// TwinCAT 3 PLC project sample_delivery
// ProgramVersion: 3.1.4023.0
// libraries:
//   LCLS Sample Delivery, * (SLAC - LCLS)
//   LCLS Vacuum, * (SLAC - LCLS)
//   Tc2_Standard, * (Beckhoff Automation GmbH)
//   Tc2_System, * (Beckhoff Automation GmbH)
//   Tc3_Module, * (Beckhoff Automation GmbH)
// project tree:
//   GVLs/ GVL_RCC.TcGVL (not stored), GVL_SDS.TcGVL
//   / PlcTask.TcTTO (not stored), SerialComm.TcTTO (not stored)
//   POUs/ MAIN.TcPOU (not stored), PRG_RCC.TcPOU, SerialTxRx.TcPOU (not stored)
// real-time tasks:
//   TASK PlcTask: cycle T#10ms, priority 20, ADS port 350
//   TASK SerialComm: cycle T#10ms, priority 1, ADS port 351
// I/O:
//   DEVICE Device 1 (EtherCAT), AmsNetId 172.21.38.25.2.1
//     Term 1 (EK1200)
//     Box 17 (EP9128-0021)
//     ALI (EP1111)
//     ALI_X (EP7041-0002)
//     ALI_Y (EP7041-0002)
//     ALI_Z (EP7041-0002)
//     ALI_X_ENC (EP5101-0011)
//     ALI_Gauges (EP3174-0002)
//     ALI_PropValve (EP7041-0002)
//     ALI_Y_ENC (EP5101-0011)
//     ALI_DIO (EP2338-0001)
//     M3 Selector A (EP1111)
//     M3 Selector A Digital IO (EP2338-1001)
//     M3 Selector A Serial IO (EP6002-0002)
//     M3 Selector B (EP1111)
//     M3 Selector B Digital IO (EP2338-1001)
//     M3 Selector B Serial IO (EP6002-0002)
//     PCM A (EP1111)
//     PCM A (EP4374-0002)
//     PCM A (EP3174-0002)
//     PCM A (EP6002-0002)
//     PCM B (EP1111)
//     PCM B (EP4374-0002)
//     PCM B (EP3174-0002)
//     PCM B (EP6002-0002)
//     Gas_Mani (EP1111)
//     Gas_Mani_NeedleValve (EP4374-0002)
//     Gas_Mani_ValveCtrl (EP2338-0001)
//     Gas_Mani_ValveRbk (EP2338-0001)
//     M3 Selector C (EP1111)
//     M3 Selector C Digital IO (EP2338-1001)
//     M3 Selector C Serial IO (EP6002-0002)
//     M3 Selector D (EP1111)
//     M3 Selector D Digital IO (EP2338-1001)
//     M3 Selector D Serial IO (EP6002-0002)
//     PCM C (EP1111)
//     PCM C (EP4374-0002)
//     PCM C (EP3174-0002)
//     PCM C (EP6002-0002)
//     PCM D (EP1111)
//     PCM D (EP4374-0002)
//     PCM D (EP3174-0002)
//     PCM D (EP6002-0002)
//     Bronkhorst MFM A
//     Bronkhorst MFM B
//     Bronkhorst MFM C
//     Bronkhorst MFM D
//     Solenoid Pair A (EP1111)
//     Solenoid Pair A Digital IO (EP2338-0001)
//     RCC A (EP1111)
//     RCC (EP2338-0001)
//     RCC_PCM_A (EP4374-0002) [EP4374-0002 2Ch. Ana. Input +/-10V, 0-10V, 0/4-20mA configurable; 2Ch. Ana. Output +/-10V, 0-10V, 0/4-20mA configurable]
// variable links:
//   sample-delivery Instance <-> Device 1 (EtherCAT)/Bronkhorst MFM A
//     PlcTask Inputs/GVL_SDS.BronkhorstA.stMFM.i_rFlow <-> TxPDO Map/fMeasure
//     PlcTask Outputs/GVL_SDS.BronkhorstA.stMFM.q_rSetpoint <-> RxPDO Map/fSetpoint
//   sample-delivery Instance <-> Device 1 (EtherCAT)/Bronkhorst MFM B
//     PlcTask Inputs/GVL_SDS.BronkhorstB.stMFM.i_rFlow <-> TxPDO Map/fMeasure
//     PlcTask Outputs/GVL_SDS.BronkhorstB.stMFM.q_rSetpoint <-> RxPDO Map/fSetpoint
//   sample-delivery Instance <-> Device 1 (EtherCAT)/Gas_Mani_ValveCtrl (EP2338-0001)
//     PlcTask Outputs/GVL_SDS.GasMan.stValve[{1..7}].qxDO <-> Channel {9..15}/Output  (7 links)
//   sample-delivery Instance <-> Device 1 (EtherCAT)/Gas_Mani_ValveRbk (EP2338-0001)
//     PlcTask Inputs/GVL_SDS.GasMan.stValve[{1..7}].ixOPN <-> Channel {1..7}/Input  (7 links)
//   sample-delivery Instance <-> Device 1 (EtherCAT)/M3 Selector A Digital IO (EP2338-1001)
//     PlcTask Outputs/GVL_SDS.M3SelectorA.stShaker01.q_xPwrDO <-> Channel 9/Output
//     PlcTask Outputs/GVL_SDS.M3SelectorA.stShaker02.q_xPwrDO <-> Channel 10/Output
//     PlcTask Outputs/GVL_SDS.M3SelectorA.stShaker03.q_xPwrDO <-> Channel 11/Output
//     PlcTask Outputs/GVL_SDS.M3SelectorA.stShaker04.q_xPwrDO <-> Channel 12/Output
//   sample-delivery Instance <-> Device 1 (EtherCAT)/M3 Selector A Serial IO (EP6002-0002)
//     SerialComm Inputs/GVL_SDS.M3SelectorA.stSensSerial.stComIn/Status <-> COM TxPDO-Map Inputs Channel 1/Status
//     SerialComm Inputs/GVL_SDS.M3SelectorA.stViciSerial.stComIn/Status <-> COM TxPDO-Map Inputs Channel 2/Status
//   sample-delivery Instance <-> Device 1 (EtherCAT)/M3 Selector B Digital IO (EP2338-1001)
//     PlcTask Outputs/GVL_SDS.M3SelectorB.stShaker01.q_xPwrDO <-> Channel 9/Output
//     PlcTask Outputs/GVL_SDS.M3SelectorB.stShaker02.q_xPwrDO <-> Channel 10/Output
//     PlcTask Outputs/GVL_SDS.M3SelectorB.stShaker03.q_xPwrDO <-> Channel 11/Output
//     PlcTask Outputs/GVL_SDS.M3SelectorB.stShaker04.q_xPwrDO <-> Channel 12/Output
//   sample-delivery Instance <-> Device 1 (EtherCAT)/M3 Selector B Serial IO (EP6002-0002)
//     SerialComm Inputs/GVL_SDS.M3SelectorB.stSensSerial.stComIn/Status <-> COM TxPDO-Map Inputs Channel 1/Status
//     SerialComm Inputs/GVL_SDS.M3SelectorB.stViciSerial.stComIn/Status <-> COM TxPDO-Map Inputs Channel 2/Status
//   sample-delivery Instance <-> Device 1 (EtherCAT)/M3 Selector C Digital IO (EP2338-1001)
//     PlcTask Outputs/GVL_SDS.M3SelectorC.stShaker01.q_xPwrDO <-> Channel 9/Output
//     PlcTask Outputs/GVL_SDS.M3SelectorC.stShaker02.q_xPwrDO <-> Channel 10/Output
//     PlcTask Outputs/GVL_SDS.M3SelectorC.stShaker03.q_xPwrDO <-> Channel 11/Output
//     PlcTask Outputs/GVL_SDS.M3SelectorC.stShaker04.q_xPwrDO <-> Channel 12/Output
//   sample-delivery Instance <-> Device 1 (EtherCAT)/M3 Selector C Serial IO (EP6002-0002)
//     SerialComm Inputs/GVL_SDS.M3SelectorC.stSensSerial.stComIn/Status <-> COM TxPDO-Map Inputs Channel 1/Status
//     SerialComm Inputs/GVL_SDS.M3SelectorC.stViciSerial.stComIn/Status <-> COM TxPDO-Map Inputs Channel 2/Status
//   sample-delivery Instance <-> Device 1 (EtherCAT)/M3 Selector D Digital IO (EP2338-1001)
//     PlcTask Outputs/GVL_SDS.M3SelectorD.stShaker01.q_xPwrDO <-> Channel 9/Output
//     PlcTask Outputs/GVL_SDS.M3SelectorD.stShaker02.q_xPwrDO <-> Channel 10/Output
//     PlcTask Outputs/GVL_SDS.M3SelectorD.stShaker03.q_xPwrDO <-> Channel 11/Output
//     PlcTask Outputs/GVL_SDS.M3SelectorD.stShaker04.q_xPwrDO <-> Channel 12/Output
//   sample-delivery Instance <-> Device 1 (EtherCAT)/M3 Selector D Serial IO (EP6002-0002)
//     SerialComm Inputs/GVL_SDS.M3SelectorD.stSensSerial.stComIn/Status <-> COM TxPDO-Map Inputs Channel 1/Status
//     SerialComm Inputs/GVL_SDS.M3SelectorD.stViciSerial.stComIn/Status <-> COM TxPDO-Map Inputs Channel 2/Status
//   sample-delivery Instance <-> Device 1 (EtherCAT)/PCM A (EP1111)
//     PlcTask Inputs/GVL_SDS.PCMA.stBaseIO.i_SyncUnitWC <-> WcState/WcState
//   sample-delivery Instance <-> Device 1 (EtherCAT)/PCM A (EP4374-0002)
//     PlcTask Inputs/GVL_SDS.PCMA.stPropAir1.i_iPressRB <-> AI Inputs Channel 1/Value
//     PlcTask Inputs/GVL_SDS.PCMA.stPropAir2.i_iPressRB <-> AI Inputs Channel 2/Value
//     PlcTask Outputs/GVL_SDS.PCMA.stPropAir1.q_iPressCt <-> AO Outputs Channel 3/Analog output
//     PlcTask Outputs/GVL_SDS.PCMA.stPropAir2.q_iPressCt <-> AO Outputs Channel 4/Analog output
//   sample-delivery Instance <-> Device 1 (EtherCAT)/PCM A (EP6002-0002)
//     SerialComm Inputs/GVL_SDS.PCMA.stSerial1.stComIn/Status <-> COM TxPDO-Map Inputs Channel 1/Status
//     SerialComm Inputs/GVL_SDS.PCMA.stSerial2.stComIn/Status <-> COM TxPDO-Map Inputs Channel 2/Status
//     SerialComm Outputs/GVL_SDS.PCMA.stSerial1.stComOut/Ctrl <-> COM RxPDO-Map Outputs Channel 1/Ctrl
//     SerialComm Outputs/GVL_SDS.PCMA.stSerial2.stComOut/Ctrl <-> COM RxPDO-Map Outputs Channel 2/Ctrl
//   sample-delivery Instance <-> Device 1 (EtherCAT)/PCM B (EP1111)
//     PlcTask Inputs/GVL_SDS.PCMB.stBaseIO.i_SyncUnitWC <-> WcState/WcState
//   sample-delivery Instance <-> Device 1 (EtherCAT)/PCM B (EP4374-0002)
//     PlcTask Inputs/GVL_SDS.PCMB.stPropAir1.i_iPressRB <-> AI Inputs Channel 1/Value
//     PlcTask Inputs/GVL_SDS.PCMB.stPropAir2.i_iPressRB <-> AI Inputs Channel 2/Value
//     PlcTask Outputs/GVL_SDS.PCMB.stPropAir1.q_iPressCt <-> AO Outputs Channel 3/Analog output
//     PlcTask Outputs/GVL_SDS.PCMB.stPropAir2.q_iPressCt <-> AO Outputs Channel 4/Analog output
//   sample-delivery Instance <-> Device 1 (EtherCAT)/PCM B (EP6002-0002)
//     SerialComm Inputs/GVL_SDS.PCMB.stSerial1.stComIn/Status <-> COM TxPDO-Map Inputs Channel 1/Status
//     SerialComm Inputs/GVL_SDS.PCMB.stSerial2.stComIn/Status <-> COM TxPDO-Map Inputs Channel 2/Status
//     SerialComm Outputs/GVL_SDS.PCMB.stSerial1.stComOut/Ctrl <-> COM RxPDO-Map Outputs Channel 1/Ctrl
//     SerialComm Outputs/GVL_SDS.PCMB.stSerial2.stComOut/Ctrl <-> COM RxPDO-Map Outputs Channel 2/Ctrl
//   sample-delivery Instance <-> Device 1 (EtherCAT)/PCM C (EP1111)
//     PlcTask Inputs/GVL_SDS.PCMC.stBaseIO.i_SyncUnitWC <-> WcState/WcState
//   sample-delivery Instance <-> Device 1 (EtherCAT)/PCM C (EP4374-0002)
//     PlcTask Inputs/GVL_SDS.PCMC.stPropAir1.i_iPressRB <-> AI Inputs Channel 1/Value
//     PlcTask Inputs/GVL_SDS.PCMC.stPropAir2.i_iPressRB <-> AI Inputs Channel 2/Value
//     PlcTask Outputs/GVL_SDS.PCMC.stPropAir1.q_iPressCt <-> AO Outputs Channel 3/Analog output
//     PlcTask Outputs/GVL_SDS.PCMC.stPropAir2.q_iPressCt <-> AO Outputs Channel 4/Analog output
//   sample-delivery Instance <-> Device 1 (EtherCAT)/PCM C (EP6002-0002)
//     SerialComm Inputs/GVL_SDS.PCMC.stSerial1.stComIn/Status <-> COM TxPDO-Map Inputs Channel 1/Status
//     SerialComm Inputs/GVL_SDS.PCMC.stSerial2.stComIn/Status <-> COM TxPDO-Map Inputs Channel 2/Status
//     SerialComm Outputs/GVL_SDS.PCMC.stSerial1.stComOut/Ctrl <-> COM RxPDO-Map Outputs Channel 1/Ctrl
//     SerialComm Outputs/GVL_SDS.PCMC.stSerial2.stComOut/Ctrl <-> COM RxPDO-Map Outputs Channel 2/Ctrl
//   sample-delivery Instance <-> Device 1 (EtherCAT)/PCM D (EP1111)
//     PlcTask Inputs/GVL_SDS.PCMD.stBaseIO.i_SyncUnitWC <-> WcState/WcState
//   sample-delivery Instance <-> Device 1 (EtherCAT)/PCM D (EP4374-0002)
//     PlcTask Inputs/GVL_SDS.PCMD.stPropAir1.i_iPressRB <-> AI Inputs Channel 1/Value
//     PlcTask Inputs/GVL_SDS.PCMD.stPropAir2.i_iPressRB <-> AI Inputs Channel 2/Value
//     PlcTask Outputs/GVL_SDS.PCMD.stPropAir1.q_iPressCt <-> AO Outputs Channel 3/Analog output
//     PlcTask Outputs/GVL_SDS.PCMD.stPropAir2.q_iPressCt <-> AO Outputs Channel 4/Analog output
//   sample-delivery Instance <-> Device 1 (EtherCAT)/PCM D (EP6002-0002)
//     SerialComm Inputs/GVL_SDS.PCMD.stSerial1.stComIn/Status <-> COM TxPDO-Map Inputs Channel 1/Status
//     SerialComm Inputs/GVL_SDS.PCMD.stSerial2.stComIn/Status <-> COM TxPDO-Map Inputs Channel 2/Status
//     SerialComm Outputs/GVL_SDS.PCMD.stSerial1.stComOut/Ctrl <-> COM RxPDO-Map Outputs Channel 1/Ctrl
//     SerialComm Outputs/GVL_SDS.PCMD.stSerial2.stComOut/Ctrl <-> COM RxPDO-Map Outputs Channel 2/Ctrl
//   sample-delivery Instance <-> Device 1 (EtherCAT)/RCC (EP2338-0001)
//     PlcTask Inputs/GVL_RCC.RCC_VRC_01.i_xOpnLS <-> Channel 1/Input
//     PlcTask Inputs/GVL_RCC.RCC_VRC_02.i_xOpnLS <-> Channel 2/Input
//     PlcTask Inputs/GVL_RCC.RCC_VRC_03.i_xOpnLS <-> Channel 3/Input
//     PlcTask Inputs/GVL_RCC.RCC_VRC_04.i_xOpnLS <-> Channel 4/Input
//     PlcTask Inputs/GVL_RCC.RCC_VRC_05.i_xOpnLS <-> Channel 5/Input
//     PlcTask Inputs/GVL_RCC.RCC_VRC_06.i_xOpnLS <-> Channel 6/Input
//     PlcTask Inputs/GVL_RCC.RCC_VRC_07.i_xOpnLS <-> Channel 7/Input
//     PlcTask Inputs/GVL_RCC.RCC_VRC_08.i_xOpnLS <-> Channel 8/Input
//     PlcTask Outputs/GVL_RCC.RCC_VRC_01.q_xOPN_DO <-> Channel 9/Output
//     PlcTask Outputs/GVL_RCC.RCC_VRC_02.q_xOPN_DO <-> Channel 10/Output
//     PlcTask Outputs/GVL_RCC.RCC_VRC_03.q_xOPN_DO <-> Channel 11/Output
//     PlcTask Outputs/GVL_RCC.RCC_VRC_04.q_xOPN_DO <-> Channel 12/Output
//     PlcTask Outputs/GVL_RCC.RCC_VRC_05.q_xOPN_DO <-> Channel 13/Output
//     PlcTask Outputs/GVL_RCC.RCC_VRC_06.q_xOPN_DO <-> Channel 14/Output
//     PlcTask Outputs/GVL_RCC.RCC_VRC_07.q_xOPN_DO <-> Channel 15/Output
//     PlcTask Outputs/GVL_RCC.RCC_VRC_08.q_xOPN_DO <-> Channel 16/Output
//   sample-delivery Instance <-> Device 1 (EtherCAT)/RCC_PCM_A (EP4374-0002)
//     PlcTask Inputs/PRG_RCC.RCC_PCM.stPropAir1.i_iPressRB <-> AI Inputs Channel 1/Value
//     PlcTask Inputs/PRG_RCC.RCC_PCM.stPropAir2.i_iPressRB <-> AI Inputs Channel 2/Value
//     PlcTask Outputs/PRG_RCC.RCC_PCM.stPropAir1.q_iPressCt <-> AO Outputs Channel 3/Analog output
//     PlcTask Outputs/PRG_RCC.RCC_PCM.stPropAir2.q_iPressCt <-> AO Outputs Channel 4/Analog output
//   sample-delivery Instance <-> Device 1 (EtherCAT)/Solenoid Pair A Digital IO (EP2338-0001)
//     PlcTask Outputs/GVL_SDS.SolenoidPairA.q_xDO1 <-> Channel 9/Output
//     PlcTask Outputs/GVL_SDS.SolenoidPairA.q_xDO2 <-> Channel 10/Output

// ---- GVLs/GVL_SDS.TcGVL
VAR_GLOBAL

// TODO: FIX Linking for Devices will be deployed
//  Working: Bronkhorst MFM B
{attribute 'pytmc' := 'pv: XCS:SDS:SEL:A'}
{attribute 'TcLinkTo' := '.stSensSerial.stComIn.Status := TIIB[M3 Selector A Serial IO (EP6002-0002)]^COM TxPDO-Map Inputs Channel 1^Status;
                          .stViciSerial.stComIn.Status := TIIB[M3 Selector A Serial IO (EP6002-0002)]^COM TxPDO-Map Inputs Channel 2^Status;
                          .stSensSerial.stComOut.Ctrl := TIID^MAIN (EtherCAT)^M3 Selector A Serial IO (EP6002-0002)^COM RxPDO-Map Outputs Channel 1^Ctrl;
                          .stViciSerial.stComOut.Ctrl := TIID^MAIN (EtherCAT)^M3 Selector A Serial IO (EP6002-0002)^COM RxPDO-Map Outputs Channel 2^Ctrl;
                          .stShaker01.q_xPwrDO := TIIB[M3 Selector A Digital IO (EP2338-1001)]^Channel 9^Output;
                          .stShaker02.q_xPwrDO := TIIB[M3 Selector A Digital IO (EP2338-1001)]^Channel 10^Output;
                          .stShaker03.q_xPwrDO := TIIB[M3 Selector A Digital IO (EP2338-1001)]^Channel 11^Output;
                          .stShaker04.q_xPwrDO := TIIB[M3 Selector A Digital IO (EP2338-1001)]^Channel 12^Output;
                          .stBaseIO.i_SyncUnitWC := TIID^MAIN (EtherCAT)^M3 Selector A (EP1111)^WcState^WcState;
                          .
'}
M3SelectorA : FB_SelectorM3;

{attribute 'pytmc' := 'pv: XCS:SDS:SEL:B'}
{attribute 'TcLinkTo' := '.stSensSerial.stComIn.Status := TIIB[M3 Selector B Serial IO (EP6002-0002)]^COM TxPDO-Map Inputs Channel 1^Status;
                          .stViciSerial.stComIn.Status := TIIB[M3 Selector B Serial IO (EP6002-0002)]^COM TxPDO-Map Inputs Channel 2^Status;
                          .stSensSerial.stComOut.Ctrl := TIID^MAIN (EtherCAT)^M3 Selector B Serial IO (EP6002-0002)^COM RxPDO-Map Outputs Channel 1^Ctrl;
                          .stViciSerial.stComOut.Ctrl := TIID^MAIN (EtherCAT)^M3 Selector B Serial IO (EP6002-0002)^COM RxPDO-Map Outputs Channel 2^Ctrl;
                          .stShaker01.q_xPwrDO := TIIB[M3 Selector B Digital IO (EP2338-1001)]^Channel 9^Output;
                          .stShaker02.q_xPwrDO := TIIB[M3 Selector B Digital IO (EP2338-1001)]^Channel 10^Output;
                          .stShaker03.q_xPwrDO := TIIB[M3 Selector B Digital IO (EP2338-1001)]^Channel 11^Output;
                          .stShaker04.q_xPwrDO := TIIB[M3 Selector B Digital IO (EP2338-1001)]^Channel 12^Output;
                          .stBaseIO.i_SyncUnitWC := TIID^MAIN (EtherCAT)^M3 Selector B (EP1111)^WcState^WcState
'}
M3SelectorB : FB_SelectorM3;

{attribute 'pytmc' := 'pv: XCS:SDS:SEL:C'}
{attribute 'TcLinkTo' := '.stSensSerial.stComIn.Status := TIIB[M3 Selector C Serial IO (EP6002-0002)]^COM TxPDO-Map Inputs Channel 1^Status;
                          .stViciSerial.stComIn.Status := TIIB[M3 Selector C Serial IO (EP6002-0002)]^COM TxPDO-Map Inputs Channel 2^Status;
                          .stSensSerial.stComOut.Ctrl := TIID^MAIN (EtherCAT)^M3 Selector C Serial IO (EP6002-0002)^COM RxPDO-Map Outputs Channel 1^Ctrl;
                          .stViciSerial.stComOut.Ctrl := TIID^MAIN (EtherCAT)^M3 Selector C Serial IO (EP6002-0002)^COM RxPDO-Map Outputs Channel 2^Ctrl;
                          .stShaker01.q_xPwrDO := TIIB[M3 Selector C Digital IO (EP2338-1001)]^Channel 9^Output;
                          .stShaker02.q_xPwrDO := TIIB[M3 Selector C Digital IO (EP2338-1001)]^Channel 10^Output;
                          .stShaker03.q_xPwrDO := TIIB[M3 Selector C Digital IO (EP2338-1001)]^Channel 11^Output;
                          .stShaker04.q_xPwrDO := TIIB[M3 Selector C Digital IO (EP2338-1001)]^Channel 12^Output;
                          .stBaseIO.i_SyncUnitWC := TIID^MAIN (EtherCAT)^M3 Selector C (EP1111)^WcState^WcState
'}
M3SelectorC : FB_SelectorM3;

{attribute 'pytmc' := 'pv: XCS:SDS:SEL:D'}
{attribute 'TcLinkTo' := '.stSensSerial.stComIn.Status := TIIB[M3 Selector D Serial IO (EP6002-0002)]^COM TxPDO-Map Inputs Channel 1^Status;
                          .stViciSerial.stComIn.Status := TIIB[M3 Selector D Serial IO (EP6002-0002)]^COM TxPDO-Map Inputs Channel 2^Status;
                          .stSensSerial.stComOut.Ctrl := TIID^MAIN (EtherCAT)^M3 Selector D Serial IO (EP6002-0002)^COM RxPDO-Map Outputs Channel 1^Ctrl;
                          .stViciSerial.stComOut.Ctrl := TIID^MAIN (EtherCAT)^M3 Selector D Serial IO (EP6002-0002)^COM RxPDO-Map Outputs Channel 2^Ctrl;
                          .stShaker01.q_xPwrDO := TIIB[M3 Selector D Digital IO (EP2338-1001)]^Channel 9^Output;
                          .stShaker02.q_xPwrDO := TIIB[M3 Selector D Digital IO (EP2338-1001)]^Channel 10^Output;
                          .stShaker03.q_xPwrDO := TIIB[M3 Selector D Digital IO (EP2338-1001)]^Channel 11^Output;
                          .stShaker04.q_xPwrDO := TIIB[M3 Selector D Digital IO (EP2338-1001)]^Channel 12^Output;
                          .stBaseIO.i_SyncUnitWC := TIID^MAIN (EtherCAT)^M3 Selector D (EP1111)^WcState^WcState
'}
M3SelectorD : FB_SelectorM3;

{attribute 'pytmc' := 'pv: XCS:SDS:PCM:A'}
{attribute 'TcLinkTo' := '.stPropAir1.i_iPressRB 	:= TIIB[PCM A (EP4374-0002)]^AI Inputs Channel 1^Value;
                          .stPropAir2.i_iPressRB 	:= TIIB[PCM A (EP4374-0002)]^AI Inputs Channel 2^Value;
                          .stPropAir1.q_iPressCt 	:= TIIB[PCM A (EP4374-0002)]^AO Outputs Channel 3^Analog output;
                          .stPropAir2.q_iPressCt 	:= TIIB[PCM A (EP4374-0002)]^AO Outputs Channel 4^Analog output;
                          .stSerial1.stComIn.Status := TIIB[PCM A (EP6002-0002)]^COM TxPDO-Map Inputs Channel 1^Status;
                          .stSerial2.stComIn.Status := TIIB[PCM A (EP6002-0002)]^COM TxPDO-Map Inputs Channel 2^Status;
                          .stSerial1.stComOut.Ctrl 	:= TIIB[PCM A (EP6002-0002)]^COM RxPDO-Map Outputs Channel 1^Ctrl;
                          .stSerial2.stComOut.Ctrl 	:= TIIB[PCM A (EP6002-0002)]^COM RxPDO-Map Outputs Channel 2^Ctrl;
                          .stBaseIO.i_SyncUnitWC 	:= TIIB[PCM A (EP1111)]^WcState^WcState;
'}
PCMA : FB_PressureControlModule;

{attribute 'pytmc' := 'pv: XCS:SDS:PCM:B'}
{attribute 'TcLinkTo' := '.stPropAir1.i_iPressRB 	:= TIIB[PCM B (EP4374-0002)]^AI Inputs Channel 1^Value;
                          .stPropAir2.i_iPressRB 	:= TIIB[PCM B (EP4374-0002)]^AI Inputs Channel 2^Value;
                          .stPropAir1.q_iPressCt 	:= TIIB[PCM B (EP4374-0002)]^AO Outputs Channel 3^Analog output;
                          .stPropAir2.q_iPressCt 	:= TIIB[PCM B (EP4374-0002)]^AO Outputs Channel 4^Analog output;
                          .stSerial1.stComIn.Status := TIIB[PCM B (EP6002-0002)]^COM TxPDO-Map Inputs Channel 1^Status;
                          .stSerial2.stComIn.Status := TIIB[PCM B (EP6002-0002)]^COM TxPDO-Map Inputs Channel 2^Status;
                          .stSerial1.stComOut.Ctrl 	:= TIIB[PCM B (EP6002-0002)]^COM RxPDO-Map Outputs Channel 1^Ctrl;
                          .stSerial2.stComOut.Ctrl 	:= TIIB[PCM B (EP6002-0002)]^COM RxPDO-Map Outputs Channel 2^Ctrl;
                          .stBaseIO.i_SyncUnitWC 	:= TIIB[PCM B (EP1111)]^WcState^WcState;
'}
PCMB : FB_PressureControlModule;

{attribute 'pytmc' := 'pv: XCS:SDS:PCM:C'}
{attribute 'TcLinkTo' := '.stPropAir1.i_iPressRB 	:= TIIB[PCM C (EP4374-0002)]^AI Inputs Channel 1^Value;
                          .stPropAir2.i_iPressRB 	:= TIIB[PCM C (EP4374-0002)]^AI Inputs Channel 2^Value;
                          .stPropAir1.q_iPressCt 	:= TIIB[PCM C (EP4374-0002)]^AO Outputs Channel 3^Analog output;
                          .stPropAir2.q_iPressCt 	:= TIIB[PCM C (EP4374-0002)]^AO Outputs Channel 4^Analog output;
                          .stSerial1.stComIn.Status := TIIB[PCM C (EP6002-0002)]^COM TxPDO-Map Inputs Channel 1^Status;
                          .stSerial2.stComIn.Status := TIIB[PCM C (EP6002-0002)]^COM TxPDO-Map Inputs Channel 2^Status;
                          .stSerial1.stComOut.Ctrl 	:= TIIB[PCM C (EP6002-0002)]^COM RxPDO-Map Outputs Channel 1^Ctrl;
                          .stSerial2.stComOut.Ctrl 	:= TIIB[PCM C (EP6002-0002)]^COM RxPDO-Map Outputs Channel 2^Ctrl;
                          .stBaseIO.i_SyncUnitWC 	:= TIIB[PCM C (EP1111)]^WcState^WcState;
                          '}
PCMC : FB_PressureControlModule;

{attribute 'pytmc' := 'pv: XCS:SDS:PCM:D'}
{attribute 'TcLinkTo' := '.stPropAir1.i_iPressRB 	:= TIIB[PCM D (EP4374-0002)]^AI Inputs Channel 1^Value;
                          .stPropAir2.i_iPressRB 	:= TIIB[PCM D (EP4374-0002)]^AI Inputs Channel 2^Value;
                          .stPropAir1.q_iPressCt 	:= TIIB[PCM D (EP4374-0002)]^AO Outputs Channel 3^Analog output;
                          .stPropAir2.q_iPressCt 	:= TIIB[PCM D (EP4374-0002)]^AO Outputs Channel 4^Analog output;
                          .stSerial1.stComIn.Status := TIIB[PCM D (EP6002-0002)]^COM TxPDO-Map Inputs Channel 1^Status;
                          .stSerial2.stComIn.Status := TIIB[PCM D (EP6002-0002)]^COM TxPDO-Map Inputs Channel 2^Status;
                          .stSerial1.stComOut.Ctrl 	:= TIIB[PCM D (EP6002-0002)]^COM RxPDO-Map Outputs Channel 1^Ctrl;
                          .stSerial2.stComOut.Ctrl 	:= TIIB[PCM D (EP6002-0002)]^COM RxPDO-Map Outputs Channel 2^Ctrl;
                          .stBaseIO.i_SyncUnitWC 	:= TIIB[PCM D (EP1111)]^WcState^WcState;
                          '}
PCMD : FB_PressureControlModule;

{attribute 'pytmc' := 'pv: XCS:SDS:MAN'}
{attribute 'TcLinkTo' := '.stValve[1].qxDO := TIIB[Gas_Mani_ValveCtrl (EP2338-0001)]^Channel 9^Output;
                          .stValve[1].ixOPN := TIIB[Gas_Mani_ValveRbk (EP2338-0001)]^Channel 1^Input;
                          .stValve[2].qxDO := TIIB[Gas_Mani_ValveCtrl (EP2338-0001)]^Channel 10^Output;
                          .stValve[2].ixOPN := TIIB[Gas_Mani_ValveRbk (EP2338-0001)]^Channel 2^Input;
                          .stValve[3].qxDO := TIIB[Gas_Mani_ValveCtrl (EP2338-0001)]^Channel 11^Output;
                          .stValve[3].ixOPN := TIIB[Gas_Mani_ValveRbk (EP2338-0001)]^Channel 3^Input;
                          .stValve[4].qxDO := TIIB[Gas_Mani_ValveCtrl (EP2338-0001)]^Channel 12^Output;
                          .stValve[4].ixOPN := TIIB[Gas_Mani_ValveRbk (EP2338-0001)]^Channel 4^Input;
                          .stValve[5].qxDO := TIIB[Gas_Mani_ValveCtrl (EP2338-0001)]^Channel 13^Output;
                          .stValve[5].ixOPN := TIIB[Gas_Mani_ValveRbk (EP2338-0001)]^Channel 5^Input;
                          .stValve[6].qxDO := TIIB[Gas_Mani_ValveCtrl (EP2338-0001)]^Channel 14^Output;
                          .stValve[6].ixOPN := TIIB[Gas_Mani_ValveRbk (EP2338-0001)]^Channel 6^Input;
                          .stValve[7].qxDO := TIIB[Gas_Mani_ValveCtrl (EP2338-0001)]^Channel 15^Output;
                          .stValve[7].ixOPN := TIIB[Gas_Mani_ValveRbk (EP2338-0001)]^Channel 7^Input;
                          .stBaseIO.i_SyncUnitWC :=	TIID^MAIN (EtherCAT)^Gas_Mani (EP1111)^WcState^WcState;
'}
GasMan : FB_GasManifold;

{attribute 'pytmc' := 'pv: XCS:SDS:MFM:A'}
{attribute 'TcLinkTo' := '.stMFM.i_rFlow := 	TIIB[Bronkhorst MFM A]^TxPDO Map^fMeasure;
                          .stMFM.q_rSetpoint := TIIB[Bronkhorst MFM A]^RxPDO Map^fSetpoint;
'}
BronkhorstA : FB_BronkhorstMFM;

{attribute 'pytmc' := 'pv: XCS:SDS:MFM:B'}
{attribute 'TcLinkTo' := '.stMFM.i_rFlow 		:= 	TIIB[Bronkhorst MFM B]^TxPDO Map^fMeasure;
                          .stMFM.q_rSetpoint 	:=  TIIB[Bronkhorst MFM B]^RxPDO Map^fSetpoint;
'}
BronkhorstB : FB_BronkhorstMFM;

{attribute 'pytmc' := 'pv: XCS:SDS:MFM:C'}
{attribute 'TcLinkTo' := '.stMFM.i_rFlow := TIID^MAIN (EtherCAT)^Bronkhorst MFM C^TxPDO Map^fMeasure;
                          .stMFM.q_rSetpoint := TIID^MAIN (EtherCAT)^Bronkhorst MFM C^RxPDO Map^fSetpoint;
'}
BronkhorstC : FB_BronkhorstMFM;

{attribute 'pytmc' := 'pv: XCS:SDS:MFM:D'}
{attribute 'TcLinkTo' := '.stMFM.i_rFlow := TIID^MAIN (EtherCAT)^Bronkhorst MFM D^TxPDO Map^fMeasure;
                          .stMFM.q_rSetpoint := TIID^MAIN (EtherCAT)^Bronkhorst MFM D^RxPDO Map^fSetpoint;
'}
BronkhorstD : FB_BronkhorstMFM;

{attribute 'pytmc' := 'pv: XCS:SDS:SPR:A'}
{attribute 'TcLinkTo' := '.q_xDO1 := TIIB[Solenoid Pair A Digital IO (EP2338-0001)]^Channel 9^Output;
                          .q_xDO2 := TIIB[Solenoid Pair A Digital IO (EP2338-0001)]^Channel 10^Output;
'}
SolenoidPairA : FB_SolenoidPair;


END_VAR

// ---- POUs/PRG_RCC.TcPOU
PROGRAM PRG_RCC
VAR

    {attribute 'pytmc' :=' pv: XCS:RCC:01'}
    stRCC_CTL_SIM : ST_RCC;
    fbRCC_SIM 	  : FB_RCC;

    {attribute 'pytmc' :=' pv: XCS:RCC:02'}
    stRCC_CTL_HPLC : ST_RCC;
    fbRCC_HPLC 	  : FB_RCC;

    RCC_GCP_01_dummy : ST_VG;
    xSystemOverrideMode_RCC : BOOL := FALSE;

    {attribute 'pytmc' := 'pv: XCS:SDS:RCC:PCM'}
    {attribute 'TcLinkTo' := '.stPropAir1.i_iPressRB 	:= TIIB[RCC_PCM_A (EP4374-0002)]^AI Inputs Channel 1^Value;
                          .stPropAir2.i_iPressRB 		:= TIIB[RCC_PCM_A (EP4374-0002)]^AI Inputs Channel 2^Value;
                          .stPropAir1.q_iPressCt 		:= TIIB[RCC_PCM_A (EP4374-0002)]^AO Outputs Channel 3^Analog output;
                          .stPropAir2.q_iPressCt 		:= TIIB[RCC_PCM_A (EP4374-0002)]^AO Outputs Channel 4^Analog output;
    '}
    RCC_PCM : FB_PressureControlModule;
END_VAR

// dummy gauge is used to allow for RCC withough gauge interlock
RCC_GCP_01_dummy.xPRESS_OK := TRUE;
stRCC_CTL_HPLC.RCC_VRC_03_OPEN_OK := TRUE;

fbRCC_SIM( stRCC_VRC_01:= RCC_VRC_01.iq_stValve,
    stRCC_VRC_02 := RCC_VRC_02.iq_stValve,
    stRCC_VRC_03 := RCC_VRC_03.iq_stValve,
    stRCC_VRC_04 := RCC_VRC_04.iq_stValve,
    stRCC_GCP_01 := RCC_GCP_01_dummy,
    stRCC_CTL := stRCC_CTL_SIM
);


fbRCC_HPLC( stRCC_VRC_01:= RCC_VRC_05.iq_stValve,
    stRCC_VRC_02 := RCC_VRC_06.iq_stValve,
    stRCC_VRC_03 := RCC_VRC_07.iq_stValve,
    stRCC_VRC_04 := RCC_VRC_08.iq_stValve,
    stRCC_GCP_01 := RCC_GCP_01_dummy,
    stRCC_CTL := stRCC_CTL_HPLC
);

RCC_VRC_01(i_xExtILK_OK := stRCC_CTL_SIM.RCC_VRC_01_OPEN_OK,
                i_xOverrideMode := xSystemOverrideMode_RCC,
                 iq_stValve=> );

RCC_VRC_02(i_xExtILK_OK := stRCC_CTL_SIM.RCC_VRC_02_OPEN_OK,
                i_xOverrideMode := xSystemOverrideMode_RCC,
                 iq_stValve=> );
RCC_VRC_03(i_xExtILK_OK := stRCC_CTL_SIM.RCC_VRC_03_OPEN_OK,
                i_xOverrideMode := xSystemOverrideMode_RCC,
                 iq_stValve=> );

RCC_VRC_04(i_xExtILK_OK := stRCC_CTL_SIM.RCC_VRC_04_OPEN_OK,
                i_xOverrideMode := xSystemOverrideMode_RCC,
                 iq_stValve=> );
RCC_VRC_05(i_xExtILK_OK := stRCC_CTL_HPLC.RCC_VRC_01_OPEN_OK,
                i_xOverrideMode := xSystemOverrideMode_RCC,
                 iq_stValve=> );

RCC_VRC_06(i_xExtILK_OK := stRCC_CTL_HPLC.RCC_VRC_02_OPEN_OK,
                i_xOverrideMode := xSystemOverrideMode_RCC,
                 iq_stValve=> );
RCC_VRC_07(i_xExtILK_OK := stRCC_CTL_HPLC.RCC_VRC_03_OPEN_OK,
                i_xOverrideMode := xSystemOverrideMode_RCC,
                 iq_stValve=> );

RCC_VRC_08(i_xExtILK_OK := stRCC_CTL_HPLC.RCC_VRC_04_OPEN_OK,
                i_xOverrideMode := xSystemOverrideMode_RCC,
                 iq_stValve=> );

END_PROGRAM
